FUNCTION_BLOCK HydraulicCylinder
VAR_INPUT
	PressureBoreSide: LREAL;
	PressureRodSide: LREAL;
	ABore: LREAL;
	ARod: LREAL;
	LoadForcePistonFL: LREAL;
	FrictionForce: LREAL;
	PistonMass: LREAL;
	par : ST_pValveControlledCylinder;
END_VAR
VAR_OUTPUT
	PistonAcceleration: LREAL;
	PistonVelocity : LREAL;
	PistonPosition : LREAL;
END_VAR
VAR
	ssMethodType : SINT := 1; 
	fbPistonVelocity : DiscreteIntegrator;
	fbPistonPosition : DiscreteIntegrator;

END_VAR


(* Outputs for Atomic SubSystem: '<Root>/HydraulicCylinder' *)
(* Outport: '<Root>/PistonAcceleration' incorporates:
 *  Gain: '<S1>/Gain1'
 *  Gain: '<S1>/Gain2'
 *  Product: '<S1>/Divide '
 *  Product: '<S1>/Product'
 *  Product: '<S1>/Product1'
 *  Sum: '<S1>/sum' *)
 
//Area Cylinder
ABore := EXPT(par.DBore,2) * (par.pi/4.0);
ARod := (EXPT(par.DBore,2) - EXPT(par.DRod,2)) * (par.pi/4.0);
 
PistonAcceleration := (((((PressureBoreSide * ABore)) - ((PressureRodSide * ARod))) - FrictionForce) - LoadForcePistonFL) / PistonMass;
(* End of Outputs for SubSystem: '<Root>/HydraulicCylinder' *)

fbPistonVelocity(
	ssMethodType := ssMethodType,
	In1 := PistonAcceleration,
	Out1 => PistonVelocity
	);
	
fbPistonPosition(
	ssMethodType := ssMethodType,
	In1 := PistonVelocity,
	Out1 => PistonPosition
	);

END_FUNCTION_BLOCK

(* stored: Version 1.1.0.1, ProductVersion 3.1.4024.9
   POU HydraulicCylinder: Id {3bf06456-7c7d-48f2-a9cc-e4b64f4dae07}, SpecialFunc None *)
